Staubli VAL3: onSave.pgx

public program onSave(string& x_sItem[])
  local num i
  local num l_nSize
  local TrajectoryItem l_tTraj
begin
  //if bToSave
  // update
  if isDefined(pt:tTraj[jEditPoint.sID])
    pt:tTraj[jEditPoint.sID]=jEditPoint
    call pt:link_it(jEditPoint.sID)
    if jEditPoint.sID=="home"
      cycleStatus:bHomeLoaded=false
    endIf
  endIf
  // saveIt
  pt:libSave()
  bToSave=false
  // endIf
end
